TEXTLIST OutputType
  0 = 'Digital'
  1 = 'PWM'
   = ''
END_TEXTLIST

(* stored: Version 1.1.0.1
   TextList OutputType: Id {c0c799cc-1bb9-4ae4-aefe-a06c1626b771} *)
